// TIA Portal V20 export
// export: Created 2026-07-16T23:20:25.8190038Z, ExportSetting WithDefaults, DisplayName Totally Integrated Automation Portal, DisplayVersion V20 Update 5, DisplayName TIA Portal Openness, DisplayVersion V20 Update 4, DisplayName TIA Portal Version Control Interface, DisplayVersion V20 Update 5, DisplayName SINAMICS Startdrive Advanced, DisplayVersion V20, DisplayName SINAMICS DCC, DisplayVersion V20, DisplayName SINAMICS Startdrive G130, G150, S120, S150, SINAMICS MV, G220, S200, S210, DisplayVersion V20, DisplayName SINAMICS Startdrive G110M, G120, G120C, G120D, G120P, G115D, DisplayVersion V20, DisplayName STEP 7 Professional, DisplayVersion V20 Update 5, DisplayName STEP 7 Safety, DisplayVersion V20 Update 2, DisplayName WinCC Basic/Comfort/Advanced, DisplayVersion V20 Update 5, DisplayName WinCC Unified, DisplayVersion V20 Update 5
TYPE "UDT_PusherIO"
// stored: IsFailsafeCompliant false
   STRUCT
      "Step" : Int;
      Fitted : Bool;
      Enable : Bool;
      Mode : Int;
      HopperHighLevel : Bool;
      ManualCycleCmd : Bool;
      ParkCmd : Bool;   // In (FC_ControlMain, from the sequencer's PusherParkCmd): plant pre-start park request - while set, an idle off-home ram reparks to home after the pre-motion warning (REQ-045). With a live cycle request, one of the only two repark occasions (owner ruling 2026-07-16); jog release deliberately leaves the ram where it stopped (REQ-039).
      CycleInhibit : Bool;   // In (FC_ControlMain, from the sequencer's PusherCycleInhibitCmd): the plant has a live stop reason - no cycle may launch (CycleRequest gated) and an in-flight cycle aborts to Retract and parks (CycleAbort). Hand-jog is deliberately exempt (owner amendment 2026-07-16, REQ-040): only the mode-0 force (stop button/unhealthy) blocks jogging.
      JogExtendCmd : Bool;
      JogRetractCmd : Bool;
      HomeLimit : Bool;
      FullTravelLimit : Bool;
      HighPressure : Bool;
      PowerPackRunningFB : Bool;
      FaultReset : Bool;
      EndTravelTimeout : Real;
      ParkedTimeout : Real;
      EndTravelHoldTime : Real;
      PumpRunOnTime : Real;
      JogWarningTime : Real;
      PressureTripConfirmTime : Real;
      PressureClearResumeDelay : Real;
      PressureTripCountThreshold : Int;
      Cycling : Bool;
      Blocked : Bool;
      EndTravelTimeoutFault : Bool;
      ParkedTimeoutFault : Bool;
      BothSwitchesFault : Bool;
      RunPowerPack : Bool;
      Extend : Bool;
      Retract : Bool;
      JogPreStartSounder : Bool;
   END_STRUCT;
END_TYPE
